/// Returns a reference to the process-global `LogManager` singleton.
///
/// The singleton is a `VAR_STAT` inside this FUNCTION — no GVL required.
///
/// Usage:
/// ```st
/// // Register an appender at startup:
/// GetLogManager().Register(my_otel_appender);
///
/// // Raise the global floor to Information:
/// GetLogManager().Level := LogLevel.Information;
/// ```
FUNCTION PUBLIC GetLogManager : REFERENCE TO LogManager
VAR_STAT
	_instance : LogManager;
END_VAR

GetLogManager REF= _instance;

END_FUNCTION

(* stored: Version 1.1.0.1
   POU GetLogManager: Id {09a0b1c2-d3e4-5678-09a0-b1c2d3e45678}, SpecialFunc None *)
